INTERFACE I_Test

METHOD M_Cyclic
VAR_INPUT
END_VAR
END_METHOD

END_INTERFACE

(* stored: Version 1.1.0.1
   Itf I_Test: Id {ef95b8a1-d886-4997-bb78-1097fcde069f}
   Method M_Cyclic: Id {b92aeb6d-534a-485e-8b6c-bcc0a806c6c2} *)
